{attribute addProperty BoxType "EL6201-0000-0017"}
{attribute addProperty Id "ASI_Inputs_DeviceAT %I*ASI_Inputs_Device_6E2FC913248310ASI_StatusAT %I*ASI_Status_A408178488110ASI_Outputs_DeviceAT %Q*ASI_Outputs_Device_4A17E548248310ASI_ControlAT %Q*ASI_Control_3C9D221D4050WcStateAT %I*WcState_98A4DF7520.250InfoDataAT %I*InfoData_BC63D37F80100"}
{attribute addProperty CRC "3564403269"}
{attribute addProperty SizeInBites "706"}
{attribute addProperty SizeInBytes "88.25"}
TYPE EL6201_E1F366A1 :
STRUCT
	{attribute addProperty Name "ASI_Inputs_Device"}
	ASI_Inputs_Device : ASI_Inputs_Device_6E2FC913;
	{attribute addProperty Name "ASI_Status"}
	ASI_Status : ASI_Status_A4081784;
	{attribute addProperty Name "ASI_Outputs_Device"}
	ASI_Outputs_Device : ASI_Outputs_Device_4A17E548;
	{attribute addProperty Name "ASI_Control"}
	ASI_Control : ASI_Control_3C9D221D;
	{attribute addProperty Name "WcState"}
	WcState : WcState_98A4DF75;
	{attribute addProperty Name "InfoData"}
	InfoData : InfoData_BC63D37F;
END_STRUCT
END_TYPE

(* stored: Version 1.2.0.0, ProductVersion 3.1.4024.9
   DUT EL6201_E1F366A1: Id {67fc8f20-5356-4252-83f3-73691b7275c0} *)
